// SIMATIC S7-200 project (STEP 7-Micro/WIN), CPU 221 REL 01.10

SYMBOL_TABLE USER1
S1               I0.0
XANH_1           Q0.0     // DEN XANH 1
VANG_1           Q0.1     // DEN VANG 1
DO_1             Q0.2     // DEN DO 1
XANH_2           Q0.3     // DEN XANH 2
VANG_2           Q0.4     // DEN VANG 2
DO_2             Q0.5     // DEN DO 2
END_SYMBOL_TABLE

ORGANIZATION_BLOCK MAIN:OB1
TITLE=PROGRAM COMMENTS
BEGIN
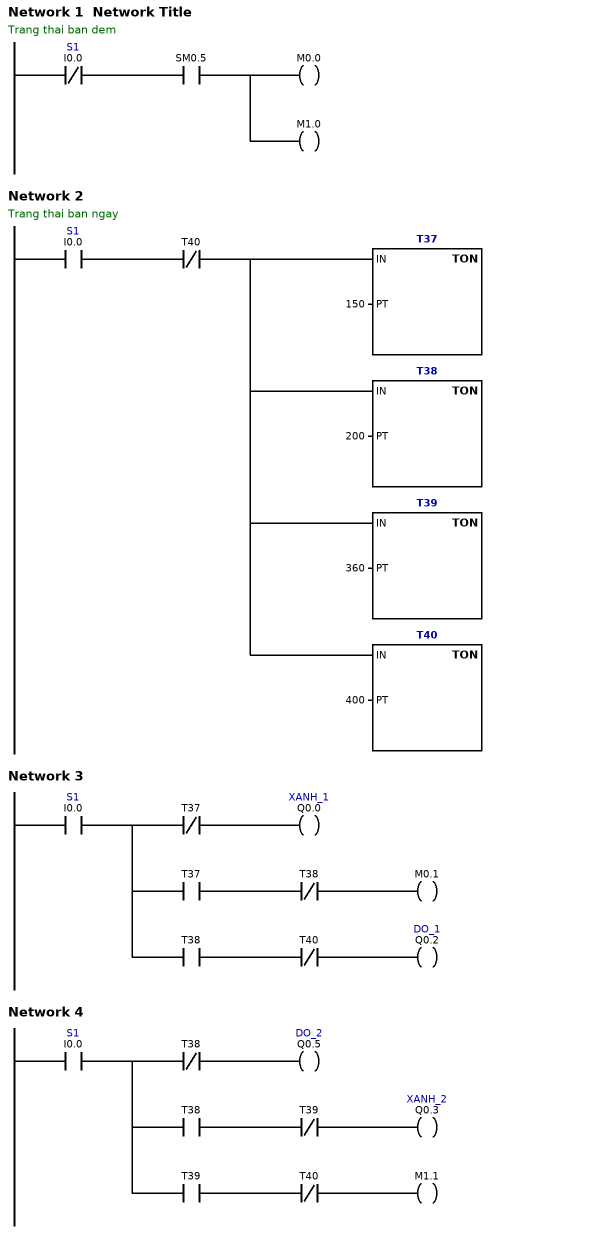
Network 1 // Network Title
// Trang thai ban dem
LDN    S1:I0.0
A      SM0.5
=      M0.0
=      M1.0
Network 2
// Trang thai ban ngay
LD     S1:I0.0
AN     T40
TON    T37, 150
TON    T38, 200
TON    T39, 360
TON    T40, 400
Network 3
LD     S1:I0.0
LPS
AN     T37
=      XANH_1:Q0.0
LRD
A      T37
AN     T38
=      M0.1
LPP
A      T38
AN     T40
=      DO_1:Q0.2
Network 4
LD     S1:I0.0
LPS
AN     T38
=      DO_2:Q0.5
LRD
A      T38
AN     T39
=      XANH_2:Q0.3
LPP
A      T39
AN     T40
=      M1.1
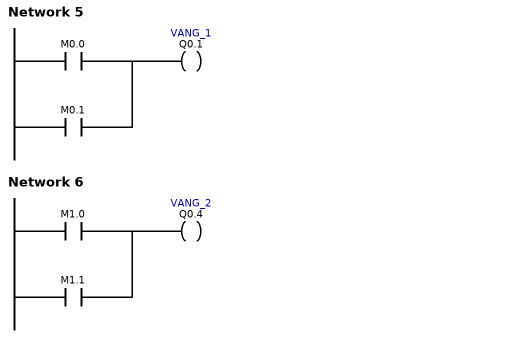
Network 5
LD     M0.0
O      M0.1
=      VANG_1:Q0.1
Network 6
LD     M1.0
O      M1.1
=      VANG_2:Q0.4
END_ORGANIZATION_BLOCK
